{attribute 'qualified_only'}
VAR_GLOBAL
	Auto	:	BOOL	:=	TRUE;
	Manual	:	BOOL	:=	FALSE;
	Off		:	BOOL	:= 	False;
END_VAR

(* stored: Version 1.1.0.1, ProductVersion 3.1.4022.10
   GVL HMI: Id {ba096bb4-055c-4569-8097-29433e5a8ad0} *)
